TYPE ST110_Recipe_t :
STRUCT
	ST110_01Y : RecipeAxisLinear2Pos_t;
	ST110_02Z : RecipeAxisLinear2Pos_t;
	ST110_03Z : RecipeAxisLinear2Pos_t;
END_STRUCT
END_TYPE

(* stored: Version 1.1.0.1, ProductVersion 3.1.4024.6
   DUT ST110_Recipe_t: Id {67830e86-a656-410c-b77d-77ee05a4605e} *)
